TYPE ST_TestSuite :
STRUCT
	nNumberOfTests : UINT;
	aTestNames : ARRAY[0..100] OF T_MaxString;
	eTestSuiteRunState : E_TestSuiteRunState := E_TestSuiteRunState.IDLE;
END_STRUCT
END_TYPE

(* stored: Version 1.1.0.1, ProductVersion 3.1.4022.12
   DUT ST_TestSuite: Id {13d3f096-dc15-407c-bd1a-874a6ea7d8e4} *)
